TYPE RealDword :
UNION
	rValue : REAL;
	dValue : DWORD;
END_UNION
END_TYPE

(* stored: Version 1.1.0.1, ProductVersion 3.1.4022.18
   DUT RealDword: Id {a8fd2386-9ff3-483e-8f92-8e75c459c97c} *)
